FUNCTION_BLOCK AB_TO_AW (* Composite FB for converting AB (BYTE) adapter to AW (WORD) adapter *)
  (* Standard: 61499-2; Description: Copyright (c) 2026 HR Agrartechnik GmbH This program and the accompanying materials are made available under the terms of the Eclipse Public License 2.0 which is available at https://www.eclipse.org/legal/epl-2.0/ SPDX-License-Identifier: EPL-2.0 *)
  (* Version 1.0, 2026-02-17, Franz Höpfinger, HR Agrartechnik GmbH *)
  PACKAGE adapter::conversion::unidirectional;
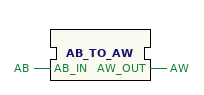
  SOCKETS
    AB_IN : adapter::types::unidirectional::AB; (* BYTE Adapter Input *)
  END_SOCKETS
  PLUGS
    AW_OUT : adapter::types::unidirectional::AW; (* WORD Adapter Output *)
  END_PLUGS
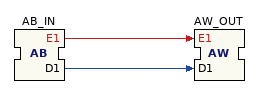
  EVENT_CONNECTIONS
    AB_IN.E1 TO AW_OUT.E1;
  END_CONNECTIONS
  DATA_CONNECTIONS
    AB_IN.D1 TO AW_OUT.D1;
  END_CONNECTIONS
END_FUNCTION_BLOCK
